{attribute addProperty BoxType "EL2911-0000-0016"}
{attribute addProperty Id "FSOEAT %Q*FSOE_C14B150F486"}
{attribute addProperty CRC "1877432700"}
{attribute addProperty SizeInBites "48"}
{attribute addProperty SizeInBytes "6"}
TYPE FSoE_Outputs_6FE7597C :
STRUCT
	{attribute addProperty Name "FSOE"}
	FSOE AT %Q* : FSOE_C14B150F;
END_STRUCT
END_TYPE

(* stored: Version 1.2.0.0, ProductVersion 3.1.4024.9
   DUT FSoE_Outputs_6FE7597C: Id {08680b8c-5ae8-4715-b305-55b81f981b5a} *)
